// TIA Portal V16 export
// export: Created 2026-06-19T14:55:51.1825097Z, ExportSetting WithDefaults, DisplayName Totally Integrated Automation Portal, DisplayVersion V16 Update 8, DisplayName TIA Portal Version Control Interface, DisplayVersion V16 Update 8, DisplayName TIA Portal Openness, DisplayVersion V16 Update 8, DisplayName SINAMICS Startdrive Advanced, DisplayVersion V16, DisplayName SINAMICS Startdrive G130, G150, S120, S150, SINAMICS MV, S210, DisplayVersion V16, DisplayName SINAMICS Startdrive G110M, G120, G120C, G120D, G120P, DisplayVersion V16, DisplayName STEP 7 Professional, DisplayVersion V16 Update 8, DisplayName STEP 7 Safety, DisplayVersion V16 Update 7, DisplayName WinCC Advanced, DisplayVersion V16 Update 8
Screen "Motor_Control"  800x480, Number=1
  ScreenLayer 
    Circle "LMP_Run" at 250,167 size 48x48
      RangeAppearanceAnimation "RangeAppearanceAnimation"
        tag Light
        0..0: back #dedbde, fore #181c31
        1..1: back #00ff00, fore #181c31
    Circle "LMP_Fault" at 400,167 size 48x48
      RangeAppearanceAnimation "RangeAppearanceAnimation"
        tag Light
        0..0: back #dedbde, fore #181c31
        1..1: back #00ff00, fore #181c31
    Button "BTN_Start" at 185,75 size 130x50  Mode=Text, TextOff="启动", TextOn="启动"
      on Press: SetBit(Tag := Button)
      on Release: ResetBit(Tag := Button)
    Button "BTN_Reset" at 493,75 size 130x50  Mode=Text, TextOff="复位", TextOn="复位"
      on Press: SetBit(Tag := Button)
      on Release: ResetBit(Tag := Button)
    Button "BTN_Stop" at 339,75 size 130x50  Mode=Text, TextOff="停止", TextOn="停止"
      on Press: SetBit(Tag := Button)
      on Release: ResetBit(Tag := Button)
    IOField "IO_Speed" at 200,245 size 180x40  DataFormat=Decimal, FormatPattern=9999999, Mode=InOutput
    SymbolicIOField "SIO_Mode" at 200,305 size 180x40  CountVisibleItems=3, Mode=InOutput, OnValue=1, TextOff="0", TextOn="1"
    TextField "TXT_Title" at 250,20 size 300x36  Text="电机控制画面"
